// TIA Portal project "Projet_Convoyeurs_S7_1200_Soluce" (V15)
// Vorlageprojekt für das Buch mit Zielsystem S7-1200

(* hardware
DEVICE "S7-1200-Station_1"  S7-1200 Station
   slot 0: "Baugruppenträger_0"  Rack  V1.0
   slot 1: "PLC_1"  CPU 1211C DC/DC/DC  6ES7 211-1AE40-0XB0  V4.1
*)

// ===== PLC "PLC_1"  CPU 1211C DC/DC/DC =====

VAR_GLOBAL   // PLC tag table "Table variables standard"
   "Convoyeur_1_1_Cellule_Debut" AT %I0.0 : Bool;
   "Convoyeur_1_1_Cellule_Fin" AT %I0.1 : Bool;
   "Convoyeur_1_2_Cellule_Debut" AT %I0.2 : Bool;
   "Convoyeur_1_2_Cellule_Fin" AT %I0.3 : Bool;
   "Convoyeur_1_3_Cellule_Debut" AT %I0.4 : Bool;
   "Convoyeur_1_3_Cellule_Fin" AT %I0.5 : Bool;
   "Convoyeur_2_1_Cellule_Debut" AT %I0.6 : Bool;
   "Convoyeur_2_1_Cellule_Fin" AT %I0.7 : Bool;
   "Convoyeur_2_2_Cellule_Debut" AT %I1.0 : Bool;
   "Convoyeur_2_2_Cellule_Fin" AT %I1.1 : Bool;
   "Convoyeur_2_3_Cellule_Debut" AT %I1.2 : Bool;
   "Convoyeur_2_3_Cellule_Fin" AT %I1.3 : Bool;
   "Convoyeur_3_1_Cellule_Debut" AT %I1.4 : Bool;
   "Convoyeur_3_1_Cellule_Fin" AT %I1.5 : Bool;
   "Convoyeur_3_2_Cellule_Debut" AT %I1.6 : Bool;
   "Convoyeur_3_2_Cellule_Fin" AT %I1.7 : Bool;
   "Convoyeur_3_3_Cellule_Debut" AT %I2.0 : Bool;
   "Convoyeur_3_3_Cellule_Fin" AT %I2.1 : Bool;
   "Convoyeur_4_1_Cellule_Debut" AT %I2.2 : Bool;
   "Convoyeur_4_1_Cellule_Fin" AT %I2.3 : Bool;
   "Convoyeur_4_2_Cellule_Debut" AT %I2.4 : Bool;
   "Convoyeur_4_2_Cellule_Fin" AT %I2.5 : Bool;
   "Convoyeur_4_3_Cellule_Debut" AT %I2.6 : Bool;
   "Convoyeur_4_3_Cellule_Fin" AT %I2.7 : Bool;
   "Convoyeur_4_4_Cellule_Debut" AT %I3.0 : Bool;
   "Convoyeur_4_4_Cellule_Fin" AT %I3.1 : Bool;
   "Convoyeur_5_1_Cellule_Debut" AT %I3.2 : Bool;
   "Convoyeur_5_1_Cellule_Fin" AT %I3.3 : Bool;
   "Convoyeur_5_2_Cellule_Debut" AT %I3.4 : Bool;
   "Convoyeur_5_2_Cellule_Fin" AT %I3.5 : Bool;
   "Convoyeur_1_1_AVANCER" AT %Q0.0 : Bool;
   "Convoyeur_1_2_AVANCER" AT %Q0.1 : Bool;
   "Convoyeur_1_3_AVANCER" AT %Q0.2 : Bool;
   "Convoyeur_2_1_AVANCER" AT %Q0.3 : Bool;
   "Convoyeur_2_2_AVANCER" AT %Q0.4 : Bool;
   "Convoyeur_2_3_AVANCER" AT %Q0.5 : Bool;
   "Convoyeur_3_1_AVANCER" AT %Q0.6 : Bool;
   "Convoyeur_3_2_AVANCER" AT %Q0.7 : Bool;
   "Convoyeur_3_3_AVANCER" AT %Q1.0 : Bool;
   "Convoyeur_4_1_AVANCER" AT %Q1.1 : Bool;
   "Convoyeur_4_2_AVANCER" AT %Q1.2 : Bool;
   "Convoyeur_4_3_AVANCER" AT %Q1.3 : Bool;
   "Convoyeur_4_4_AVANCER" AT %Q1.4 : Bool;
   "Convoyeur_5_1_AVANCER" AT %Q1.5 : Bool;
   "Convoyeur_5_2_AVANCER" AT %Q1.6 : Bool;
   "Convoyeur_5_3_AVANCER" AT %Q1.7 : Bool;
   "Convoyeur_5_4_AVANCER" AT %Q2.0 : Bool;
   "Table_1_4_AVANCER" AT %Q2.1 : Bool;
   "Table_1_4_TOURNER_DROITE" AT %Q2.2 : Bool;
   "Table_1_4_TOURNER_GAUCHE" AT %Q2.3 : Bool;
   "Table_1_5_AVANCER" AT %Q2.4 : Bool;
   "Table_1_5_TOURNER_DROITE" AT %Q2.5 : Bool;
   "Table_1_5_TOURNER_GAUCHE" AT %Q2.6 : Bool;
   "Table_2_4_AVANCER" AT %Q2.7 : Bool;
   "Table_2_4_TOURNER_DROITE" AT %Q3.0 : Bool;
   "Table_2_4_TOURNER_GAUCHE" AT %Q3.1 : Bool;
   "Table_2_5_AVANCER" AT %Q3.2 : Bool;
   "Table_2_5_TOURNER_DROITE" AT %Q3.3 : Bool;
   "Table_2_5_TOURNER_GAUCHE" AT %Q3.4 : Bool;
   "Table_3_4_AVANCER" AT %Q3.5 : Bool;
   "Table_3_4_TOURNER_GAUCHE" AT %Q3.7 : Bool;
   "Table_3_4_TOURNER_DROITE" AT %Q3.6 : Bool;
   "Table_3_5_AVANCER" AT %Q4.0 : Bool;
   "Table_3_5_TOURNER_DROITE" AT %Q4.1 : Bool;
   "Table_3_5_TOURNER_GAUCHE" AT %Q4.2 : Bool;
   "Convoyeur_5_3_Cellule_Debut" AT %I3.6 : Bool;
   "Convoyeur_5_3_Cellule_Fin" AT %I3.7 : Bool;
   "Convoyeur_5_4_Cellule_Debut" AT %I4.0 : Bool;
   "Convoyeur_5_4_Cellule_Fin" AT %I4.1 : Bool;
   "Table_1_4_Capteur_Fin" AT %I4.2 : Bool;
   "Table_1_4_Capteur_Droite" AT %I4.3 : Bool;
   "Table_1_4_Capteur_Gauche" AT %I4.4 : Bool;
   "Table_1_5_Capteur_Fin" AT %I4.5 : Bool;
   "Table_1_5_Capteur_Droite" AT %I4.6 : Bool;
   "Table_1_5_Capteur_Gauche" AT %I4.7 : Bool;
   "Table_2_4_Capteur_Fin" AT %I5.0 : Bool;
   "Table_2_4_Capteur_Droite" AT %I5.1 : Bool;
   "Table_2_4_Capteur_Gauche" AT %I5.2 : Bool;
   "Table_2_5_Capteur_Fin" AT %I5.3 : Bool;
   "Table_2_5_Capteur_Droite" AT %I5.4 : Bool;
   "Table_2_5_Capteur_Gauche" AT %I5.5 : Bool;
   "Table_3_4_Capteur_Fin" AT %I5.6 : Bool;
   "Table_3_4_Capteur_Droite" AT %I5.7 : Bool;
   "Table_3_4_Capteur_Gauche" AT %I6.0 : Bool;
   "Table_3_5_Capteur_Fin" AT %I6.1 : Bool;
   "Table_3_5_Capteur_Droite" AT %I6.2 : Bool;
   "Table_3_5_Capteur_Gauche" AT %I6.3 : Bool;
   "Nombre_Total_Ligne_1" AT %QW50 : Int;
   "Nombre_Total_Ligne_2" AT %QW52 : Int;
   "Nombre_Total_Ligne_3" AT %QW54 : Int;
   "Nombre_Total_Ligne_4" AT %QW56 : Int;
   "Nombre_Total_Ligne_5" AT %QW58 : Int;
END_VAR

// folder: DB_Convoyeurs

DATA_BLOCK "Convoyeur_1_1"   // DB3
{ S7_Optimized_Access := 'TRUE' }
VERSION : 0.1
// stored: InstanceOfName Commande_Convoyeur
"Commande_Convoyeur"
BEGIN
END_DATA_BLOCK

DATA_BLOCK "Convoyeur_1_2"   // DB4
{ S7_Optimized_Access := 'TRUE' }
VERSION : 0.1
// stored: InstanceOfName Commande_Convoyeur
"Commande_Convoyeur"
BEGIN
END_DATA_BLOCK

DATA_BLOCK "Convoyeur_4_3"   // DB5
{ S7_Optimized_Access := 'TRUE' }
VERSION : 0.1
// stored: InstanceOfName Commande_Convoyeur
"Commande_Convoyeur"
BEGIN
END_DATA_BLOCK

DATA_BLOCK "Convoyeur_1_3"   // DB6
{ S7_Optimized_Access := 'TRUE' }
VERSION : 0.1
// stored: InstanceOfName Commande_Convoyeur
"Commande_Convoyeur"
BEGIN
END_DATA_BLOCK

DATA_BLOCK "Convoyeur_4_4"   // DB7
{ S7_Optimized_Access := 'TRUE' }
VERSION : 0.1
// stored: InstanceOfName Commande_Convoyeur
"Commande_Convoyeur"
BEGIN
END_DATA_BLOCK

DATA_BLOCK "Convoyeur_5_4"   // DB8
{ S7_Optimized_Access := 'TRUE' }
VERSION : 0.1
// stored: InstanceOfName Commande_Convoyeur
"Commande_Convoyeur"
BEGIN
END_DATA_BLOCK

DATA_BLOCK "Convoyeur_5_3"   // DB9
{ S7_Optimized_Access := 'TRUE' }
VERSION : 0.1
// stored: InstanceOfName Commande_Convoyeur
"Commande_Convoyeur"
BEGIN
END_DATA_BLOCK

DATA_BLOCK "Convoyeur_2_1"   // DB10
{ S7_Optimized_Access := 'TRUE' }
VERSION : 0.1
// stored: InstanceOfName Commande_Convoyeur
"Commande_Convoyeur"
BEGIN
END_DATA_BLOCK

DATA_BLOCK "Convoyeur_2_2"   // DB12
{ S7_Optimized_Access := 'TRUE' }
VERSION : 0.1
// stored: InstanceOfName Commande_Convoyeur
"Commande_Convoyeur"
BEGIN
END_DATA_BLOCK

DATA_BLOCK "Convoyeur_2_3"   // DB14
{ S7_Optimized_Access := 'TRUE' }
VERSION : 0.1
// stored: InstanceOfName Commande_Convoyeur
"Commande_Convoyeur"
BEGIN
END_DATA_BLOCK

DATA_BLOCK "Convoyeur_4_2"   // DB15
{ S7_Optimized_Access := 'TRUE' }
VERSION : 0.1
// stored: InstanceOfName Commande_Convoyeur
"Commande_Convoyeur"
BEGIN
END_DATA_BLOCK

DATA_BLOCK "Convoyeur_5_2"   // DB16
{ S7_Optimized_Access := 'TRUE' }
VERSION : 0.1
// stored: InstanceOfName Commande_Convoyeur
"Commande_Convoyeur"
BEGIN
END_DATA_BLOCK

DATA_BLOCK "Convoyeur_3_1"   // DB19
{ S7_Optimized_Access := 'TRUE' }
VERSION : 0.1
// stored: InstanceOfName Commande_Convoyeur
"Commande_Convoyeur"
BEGIN
END_DATA_BLOCK

DATA_BLOCK "Convoyeur_3_2"   // DB20
{ S7_Optimized_Access := 'TRUE' }
VERSION : 0.1
// stored: InstanceOfName Commande_Convoyeur
"Commande_Convoyeur"
BEGIN
END_DATA_BLOCK

DATA_BLOCK "Convoyeur_3_3"   // DB21
{ S7_Optimized_Access := 'TRUE' }
VERSION : 0.1
// stored: InstanceOfName Commande_Convoyeur
"Commande_Convoyeur"
BEGIN
END_DATA_BLOCK

DATA_BLOCK "Convoyeur_4_1"   // DB22
{ S7_Optimized_Access := 'TRUE' }
VERSION : 0.1
// stored: InstanceOfName Commande_Convoyeur
"Commande_Convoyeur"
BEGIN
END_DATA_BLOCK

DATA_BLOCK "Convoyeur_5_1"   // DB23
{ S7_Optimized_Access := 'TRUE' }
VERSION : 0.1
// stored: InstanceOfName Commande_Convoyeur
"Commande_Convoyeur"
BEGIN
END_DATA_BLOCK

// folder: DB_Tables

DATA_BLOCK "Table_1_4"   // DB1
{ S7_Optimized_Access := 'TRUE' }
VERSION : 0.1
// stored: InstanceOfName Commande_Table
"Commande_Table"
BEGIN
END_DATA_BLOCK

DATA_BLOCK "Table_1_5"   // DB2
{ S7_Optimized_Access := 'TRUE' }
VERSION : 0.1
// stored: InstanceOfName Commande_Table
"Commande_Table"
BEGIN
END_DATA_BLOCK

DATA_BLOCK "Table_2_4"   // DB11
{ S7_Optimized_Access := 'TRUE' }
VERSION : 0.1
// stored: InstanceOfName Commande_Table
"Commande_Table"
BEGIN
END_DATA_BLOCK

DATA_BLOCK "Table_2_5"   // DB13
{ S7_Optimized_Access := 'TRUE' }
VERSION : 0.1
// stored: InstanceOfName Commande_Table
"Commande_Table"
BEGIN
END_DATA_BLOCK

DATA_BLOCK "Table_3_4"   // DB17
{ S7_Optimized_Access := 'TRUE' }
VERSION : 0.1
// stored: InstanceOfName Commande_Table
"Commande_Table"
BEGIN
END_DATA_BLOCK

DATA_BLOCK "Table_3_5"   // DB18
{ S7_Optimized_Access := 'TRUE' }
VERSION : 0.1
// stored: InstanceOfName Commande_Table
"Commande_Table"
BEGIN
END_DATA_BLOCK

// folder: (top level)

FUNCTION_BLOCK "Commande_Table"   // FB1, LAD
{ S7_Optimized_Access := 'TRUE' }
VERSION : 0.1
   VAR_INPUT
      Arrivee_Gauche : Bool;
      Arrivee_Droite : Bool;
      Capteur_Gauche : Bool;
      Capteur_Droite : Bool;
      Capteur_Fin_Table : Bool;
      Evacuation_en_service : Bool;
      Capteur_Debut_Convoyeur_Aval_Gauche : Bool;
      Capteur_Debut_Convoyeur_Aval_Droite : Bool;
   END_VAR
   VAR_OUTPUT
      TOURNER_GAUCHE : Bool;
      TOURNER_DROITE : Bool;
      AVANCER : Bool;
   END_VAR
   VAR
      Etape_GRAFCET : Int;
      Occupee : Bool;
      Priorite_Gauche : Bool;
   END_VAR
BEGIN

REGION Network 1 (SCL): GRAFCET de controle de la table tournante
   CASE #Etape_GRAFCET OF
       0:  // Attente arrivée d'une caisse soit à gauche soit à droite
           IF (#Arrivee_Gauche AND ((NOT #Arrivee_Droite) OR (#Arrivee_Droite AND #Priorite_Gauche))) THEN
               #Etape_GRAFCET := 1;
           END_IF;
           IF (#Arrivee_Droite AND ((NOT #Arrivee_Gauche) OR (#Arrivee_Gauche AND (NOT #Priorite_Gauche)))) THEN
               #Etape_GRAFCET := 2;
           END_IF;
       1:  // Tourner vers la gauche
           IF #Capteur_Gauche THEN
               #Etape_GRAFCET := 3;
           END_IF;
       2:  // Tourner vers la droite
           IF #Capteur_Droite THEN
               #Etape_GRAFCET := 3;
           END_IF;
       3:  // Avance de la caisse jusqu'à la fin de la table
           IF (#Capteur_Fin_Table AND (NOT #Evacuation_en_service)) THEN
               #Etape_GRAFCET := 4;
           END_IF;
           IF (#Capteur_Fin_Table AND #Evacuation_en_service) THEN
               #Etape_GRAFCET := 5;
           END_IF;
       4:  // Arrêt et Attente évacuation en service
           IF #Evacuation_en_service THEN
               #Etape_GRAFCET := 5;
           END_IF;
       5:  // Evacuation de la caisse
           IF (NOT #Capteur_Fin_Table) THEN
               #Etape_GRAFCET := 6;
           END_IF;
       6:  // Fin Evacuation de la caisse
           IF ((#Capteur_Gauche AND (NOT #Capteur_Debut_Convoyeur_Aval_Gauche)) OR (#Capteur_Droite AND (NOT #Capteur_Debut_Convoyeur_Aval_Droite))) THEN
               #Etape_GRAFCET := 0;
           END_IF;
       ELSE
           #Etape_GRAFCET := 0;
   END_CASE;
END_REGION

REGION Network 2: Commande des sorties
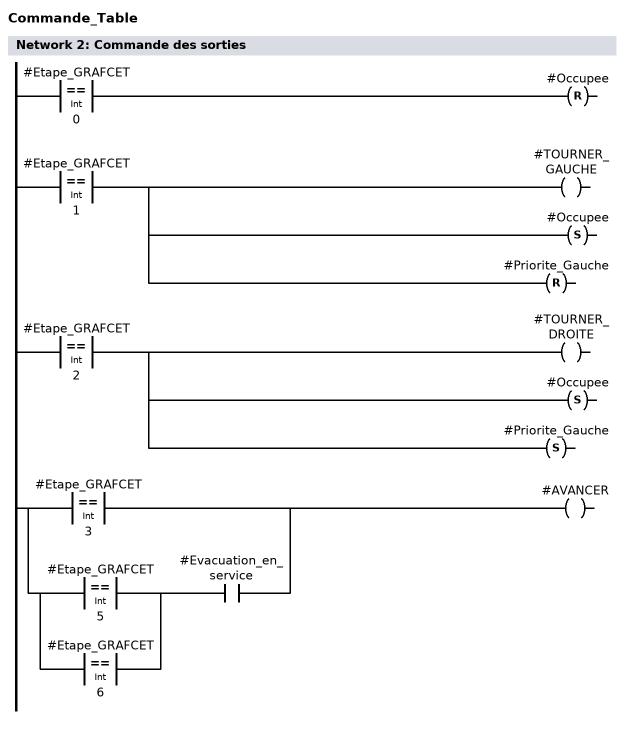
   RUNG wire#powerrail
      { S7_Templates := "SrcType := Int" } EQ_Contact(in1 := #Etape_GRAFCET, in2 := 0)
      R_Coil( #Occupee )
   END_RUNG
   RUNG wire#powerrail
      { S7_Templates := "SrcType := Int" } EQ_Contact(in1 := #Etape_GRAFCET, in2 := 1)
      wire#w1
      Coil( #TOURNER_GAUCHE )
   END_RUNG
   RUNG wire#w1
      S_Coil( #Occupee )
   END_RUNG
   RUNG wire#w1
      R_Coil( #Priorite_Gauche )
   END_RUNG
   RUNG wire#powerrail
      { S7_Templates := "SrcType := Int" } EQ_Contact(in1 := #Etape_GRAFCET, in2 := 2)
      wire#w2
      Coil( #TOURNER_DROITE )
   END_RUNG
   RUNG wire#w2
      S_Coil( #Occupee )
   END_RUNG
   RUNG wire#w2
      S_Coil( #Priorite_Gauche )
   END_RUNG
   RUNG wire#powerrail
      { S7_Templates := "SrcType := Int" } EQ_Contact(in1 := #Etape_GRAFCET, in2 := 3)
      wire#w3
      Coil( #AVANCER )
   END_RUNG
   RUNG wire#powerrail
      { S7_Templates := "SrcType := Int" } EQ_Contact(in1 := #Etape_GRAFCET, in2 := 5)
      wire#w4
      Contact( #Evacuation_en_service )
   END_RUNG wire#w3
   RUNG wire#powerrail
      { S7_Templates := "SrcType := Int" } EQ_Contact(in1 := #Etape_GRAFCET, in2 := 6)
   END_RUNG wire#w4
   // the same network as SCL:
   IF #Etape_GRAFCET = 0 THEN #Occupee := FALSE; END_IF;
   #TOURNER_GAUCHE := #Etape_GRAFCET = 1;
   IF #TOURNER_GAUCHE THEN
       #Occupee := TRUE;
       #Priorite_Gauche := FALSE;
   END_IF;
   #TOURNER_DROITE := #Etape_GRAFCET = 2;
   IF #TOURNER_DROITE THEN
       #Occupee := TRUE;
       #Priorite_Gauche := TRUE;
   END_IF;
   #AVANCER := (#Etape_GRAFCET = 3) OR (((#Etape_GRAFCET = 5) OR (#Etape_GRAFCET = 6)) AND #Evacuation_en_service);
END_REGION
END_FUNCTION_BLOCK

FUNCTION_BLOCK "Commande_Convoyeur"   // FB2, LAD
{ S7_Optimized_Access := 'TRUE' }
VERSION : 0.1
   VAR_INPUT
      Capteur_Debut_Convoyeur : Bool;
      Capteur_Fin_Convoyeur : Bool;
      Etape_Grafcet_Table : Int;
      Table_Bonne_Direction : Bool;
      Fin_Table_Amont : Bool;
      Terminaison : Bool;
   END_VAR
   VAR_OUTPUT
      AVANCER : Bool;
   END_VAR
   VAR
      Etape_GRAFCET : Int;
      Nombre_Caisses : Int;
      Nombre_Caisses_Total : Int;
      Front_Capteur_Debut : Bool;
      Front_Capteur_Fin : Bool;
   END_VAR
   VAR_TEMP   // added for the SCL form of the ladder/FBD networks
      _w1 : Bool;
      _w2 : Bool;
   END_VAR
BEGIN

REGION Network 1: Comptage Caisses
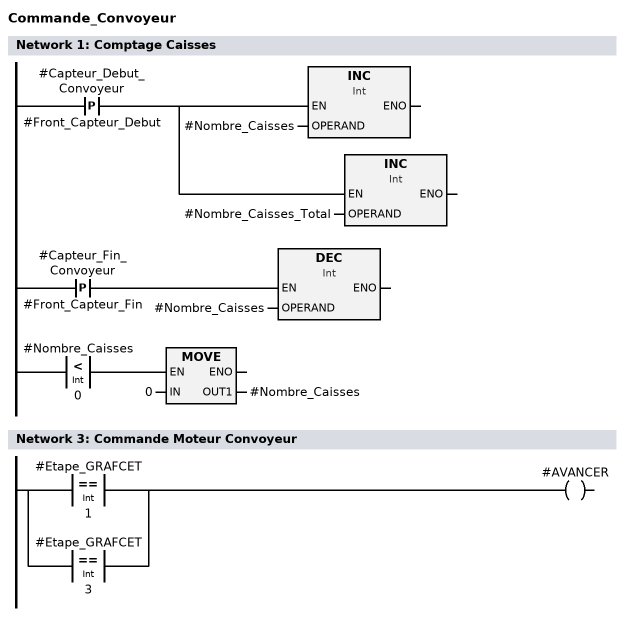
   RUNG wire#powerrail
      P_Contact(operand := #Capteur_Debut_Convoyeur, bit := #Front_Capteur_Debut)
      wire#w1
      { S7_Templates := "DestType := Int" } Inc( #Nombre_Caisses )
   END_RUNG
   RUNG wire#w1
      { S7_Templates := "DestType := Int" } Inc( #Nombre_Caisses_Total )
   END_RUNG
   RUNG wire#powerrail
      P_Contact(operand := #Capteur_Fin_Convoyeur, bit := #Front_Capteur_Fin)
      { S7_Templates := "DestType := Int" } Dec( #Nombre_Caisses )
   END_RUNG
   RUNG wire#powerrail
      { S7_Templates := "SrcType := Int" } LT_Contact(in1 := #Nombre_Caisses, in2 := 0)
      Move(in := 0, out1 => #Nombre_Caisses)
   END_RUNG
   // the same network as SCL:
   #_w1 := #Capteur_Debut_Convoyeur AND NOT #Front_Capteur_Debut;   // rising edge of #Capteur_Debut_Convoyeur
   #Front_Capteur_Debut := #Capteur_Debut_Convoyeur;
   IF #_w1 THEN
       #Nombre_Caisses := #Nombre_Caisses + 1;
       #Nombre_Caisses_Total := #Nombre_Caisses_Total + 1;
   END_IF;
   #_w2 := #Capteur_Fin_Convoyeur AND NOT #Front_Capteur_Fin;   // rising edge of #Capteur_Fin_Convoyeur
   #Front_Capteur_Fin := #Capteur_Fin_Convoyeur;
   IF #_w2 THEN #Nombre_Caisses := #Nombre_Caisses - 1; END_IF;
   IF #Nombre_Caisses < 0 THEN #Nombre_Caisses := 0; END_IF;
END_REGION

REGION Network 2 (SCL): GRAFCET de controle d'un convoyeur
   CASE #Etape_GRAFCET OF
       0:  // Attente ordre départ
           IF ((#Nombre_Caisses>0) OR ((#Nombre_Caisses=0)AND #Fin_Table_Amont))  THEN
               #Etape_GRAFCET := 1;
           END_IF;
       1:  // Avance jusqu'au capteur de fin
           IF #Capteur_Fin_Convoyeur THEN
               #Etape_GRAFCET := 2;
           END_IF;
       2:  // Arret - Attente table bonne direction et Debut chargement table
           IF (#Table_Bonne_Direction AND (#Etape_Grafcet_Table = 3)) THEN
               #Etape_GRAFCET := 3;
           END_IF;
       3:  // Avance jusqu'à chargement table terminé
           IF (NOT #Capteur_Fin_Convoyeur) THEN
               #Etape_GRAFCET := 4;
           END_IF;
       4:  // Arret - Attente fin évacuation table
           IF ((#Table_Bonne_Direction AND (#Etape_Grafcet_Table = 6))OR #Terminaison) THEN
               #Etape_GRAFCET := 0;
           END_IF;
       ELSE  
           #Etape_GRAFCET := 0;
   END_CASE;
END_REGION

REGION Network 3: Commande Moteur Convoyeur
   RUNG wire#powerrail
      { S7_Templates := "SrcType := Int" } EQ_Contact(in1 := #Etape_GRAFCET, in2 := 1)
      wire#w1
      Coil( #AVANCER )
   END_RUNG
   RUNG wire#powerrail
      { S7_Templates := "SrcType := Int" } EQ_Contact(in1 := #Etape_GRAFCET, in2 := 3)
   END_RUNG wire#w1
   // the same network as SCL:
   #AVANCER := (#Etape_GRAFCET = 1) OR (#Etape_GRAFCET = 3);
END_REGION
END_FUNCTION_BLOCK

FUNCTION "MHJ-PLC-Lab-Function-S71200" : Void   // FC9000, SCL
{ S7_Optimized_Access := 'TRUE' }
VERSION : 0.1
   VAR_TEMP
      rdTimeReturn : Int;
      outputTime : DTL;
      SyncVal : Byte;
      forVal : Int;
      forVal_2 : Int;
      Value : Byte;
   END_VAR
   VAR CONSTANT
      CompVal : Byte := 16#34;
      Value_01 : Byte := 16#11;
      Value_01_DW : DWord := 16#A165_D992;
      Value_02_DW : DWord := 16#58BE_4401;
   END_VAR
BEGIN

   #Value:=PEEK(area := 16#82,
        dbNumber := 0,
        byteOffset := 511);
   #Value := #Value + 1;

   POKE(area := 16#82,
        dbNumber := 0,
        byteOffset := 511,
        value := #Value);

   POKE(area:=16#81,
        dbNumber:=0,
        byteOffset:=1016,
        value:=#Value_01_DW);
   POKE(area := 16#81,
        dbNumber := 0,
        byteOffset := 1020,
        value := #Value_02_DW);

   POKE(area := 16#81,
        dbNumber := 0,
        byteOffset := 511,
        value := B#16#00);

   FOR #forVal := 0 TO 120 DO
       FOR #forVal_2:=0 TO 10 DO
           #rdTimeReturn:=RD_SYS_T(#outputTime);
           #rdTimeReturn := WR_SYS_T(#outputTime);
           #rdTimeReturn := RD_SYS_T(#outputTime);
           #rdTimeReturn := WR_SYS_T(#outputTime);
       END_FOR;
       #SyncVal:= PEEK(area := 16#81,
                      dbNumber := 0,
                      byteOffset := 511);
       IF #SyncVal = #CompVal THEN
          GOTO M_1;
       END_IF;
   END_FOR;
   RETURN;

   M_1:
   POKE(area := 16#81,
        dbNumber := 0,
        byteOffset := 511,
        value := B#16#0);
END_FUNCTION

ORGANIZATION_BLOCK "Main"   // OB1, LAD, ProgramCycle
TITLE = "Main Program Sweep (Cycle)"
{ S7_Optimized_Access := 'TRUE' }
VERSION : 0.1
   VAR_INPUT
      Initial_Call : Bool;   // Initial call of this OB
      Remanence : Bool;   // =True, if remanent data are available
   END_VAR
BEGIN

REGION Network 1: Konnektierungsbaustein für PLC-Lab / Appel Fonction MHJ pour Factory-IO
   // Im Netzwerk 1 wird der Konnektierungsbaustein für PLC-Lab aufgerufen.
   // Dieser Aufruf darf nicht entfernt werden!
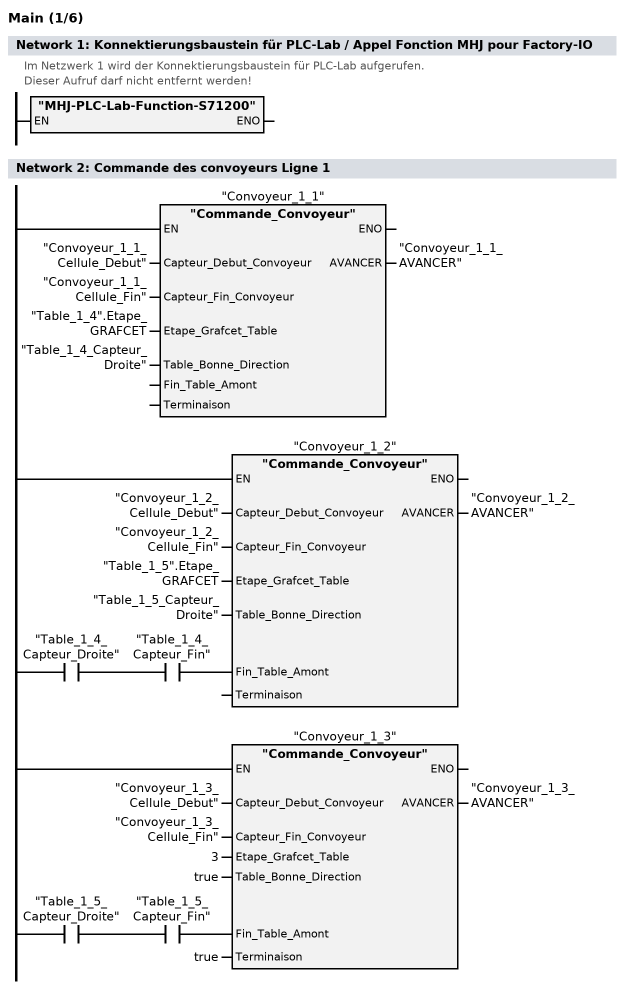
   RUNG wire#powerrail
      "MHJ-PLC-Lab-Function-S71200"()
   END_RUNG
   // the same network as SCL:
   "MHJ-PLC-Lab-Function-S71200"();
END_REGION

REGION Network 2: Commande des convoyeurs Ligne 1
   RUNG wire#powerrail
      "Convoyeur_1_1"(Capteur_Debut_Convoyeur := "Convoyeur_1_1_Cellule_Debut", Capteur_Fin_Convoyeur := "Convoyeur_1_1_Cellule_Fin", Etape_Grafcet_Table := "Table_1_4".Etape_GRAFCET, Table_Bonne_Direction := "Table_1_4_Capteur_Droite", Fin_Table_Amont :=, Terminaison :=, AVANCER => "Convoyeur_1_1_AVANCER")
   END_RUNG
   RUNG wire#powerrail
      "Convoyeur_1_2"(Fin_Table_Amont := wire#w1, Capteur_Debut_Convoyeur := "Convoyeur_1_2_Cellule_Debut", Capteur_Fin_Convoyeur := "Convoyeur_1_2_Cellule_Fin", Etape_Grafcet_Table := "Table_1_5".Etape_GRAFCET, Table_Bonne_Direction := "Table_1_5_Capteur_Droite", Terminaison :=, AVANCER => "Convoyeur_1_2_AVANCER")
   END_RUNG
   RUNG wire#powerrail
      Contact( "Table_1_4_Capteur_Droite" )
      Contact( "Table_1_4_Capteur_Fin" )
   END_RUNG wire#w1
   RUNG wire#powerrail
      "Convoyeur_1_3"(Fin_Table_Amont := wire#w2, Capteur_Debut_Convoyeur := "Convoyeur_1_3_Cellule_Debut", Capteur_Fin_Convoyeur := "Convoyeur_1_3_Cellule_Fin", Etape_Grafcet_Table := 3, Table_Bonne_Direction := true, Terminaison := true, AVANCER => "Convoyeur_1_3_AVANCER")
   END_RUNG
   RUNG wire#powerrail
      Contact( "Table_1_5_Capteur_Droite" )
      Contact( "Table_1_5_Capteur_Fin" )
   END_RUNG wire#w2
   // the same network as SCL:
   "Convoyeur_1_1"(Capteur_Debut_Convoyeur := "Convoyeur_1_1_Cellule_Debut",   // "Commande_Convoyeur"
                   Capteur_Fin_Convoyeur := "Convoyeur_1_1_Cellule_Fin",
                   Etape_Grafcet_Table := "Table_1_4".Etape_GRAFCET,
                   Table_Bonne_Direction := "Table_1_4_Capteur_Droite",
                   AVANCER => "Convoyeur_1_1_AVANCER");
   "Convoyeur_1_2"(Capteur_Debut_Convoyeur := "Convoyeur_1_2_Cellule_Debut",   // "Commande_Convoyeur"
                   Capteur_Fin_Convoyeur := "Convoyeur_1_2_Cellule_Fin",
                   Etape_Grafcet_Table := "Table_1_5".Etape_GRAFCET,
                   Table_Bonne_Direction := "Table_1_5_Capteur_Droite",
                   Fin_Table_Amont := "Table_1_4_Capteur_Droite" AND "Table_1_4_Capteur_Fin",
                   AVANCER => "Convoyeur_1_2_AVANCER");
   "Convoyeur_1_3"(Capteur_Debut_Convoyeur := "Convoyeur_1_3_Cellule_Debut",   // "Commande_Convoyeur"
                   Capteur_Fin_Convoyeur := "Convoyeur_1_3_Cellule_Fin",
                   Etape_Grafcet_Table := 3,
                   Table_Bonne_Direction := true,
                   Fin_Table_Amont := "Table_1_5_Capteur_Droite" AND "Table_1_5_Capteur_Fin",
                   Terminaison := true,
                   AVANCER => "Convoyeur_1_3_AVANCER");
END_REGION

REGION Network 3: Commande des convoyeurs Ligne 2
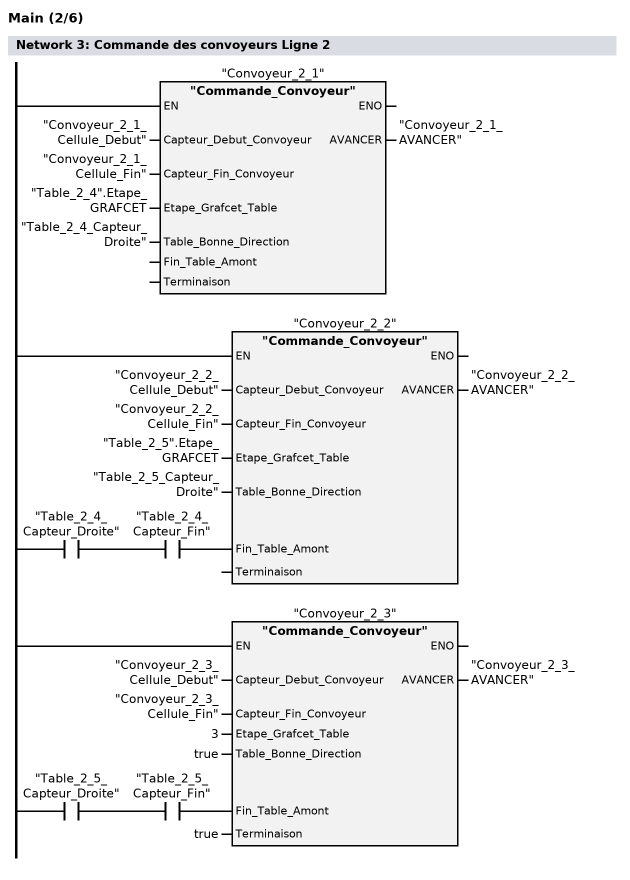
   RUNG wire#powerrail
      "Convoyeur_2_1"(Capteur_Debut_Convoyeur := "Convoyeur_2_1_Cellule_Debut", Capteur_Fin_Convoyeur := "Convoyeur_2_1_Cellule_Fin", Etape_Grafcet_Table := "Table_2_4".Etape_GRAFCET, Table_Bonne_Direction := "Table_2_4_Capteur_Droite", Fin_Table_Amont :=, Terminaison :=, AVANCER => "Convoyeur_2_1_AVANCER")
   END_RUNG
   RUNG wire#powerrail
      "Convoyeur_2_2"(Fin_Table_Amont := wire#w1, Capteur_Debut_Convoyeur := "Convoyeur_2_2_Cellule_Debut", Capteur_Fin_Convoyeur := "Convoyeur_2_2_Cellule_Fin", Etape_Grafcet_Table := "Table_2_5".Etape_GRAFCET, Table_Bonne_Direction := "Table_2_5_Capteur_Droite", Terminaison :=, AVANCER => "Convoyeur_2_2_AVANCER")
   END_RUNG
   RUNG wire#powerrail
      Contact( "Table_2_4_Capteur_Droite" )
      Contact( "Table_2_4_Capteur_Fin" )
   END_RUNG wire#w1
   RUNG wire#powerrail
      "Convoyeur_2_3"(Fin_Table_Amont := wire#w2, Capteur_Debut_Convoyeur := "Convoyeur_2_3_Cellule_Debut", Capteur_Fin_Convoyeur := "Convoyeur_2_3_Cellule_Fin", Etape_Grafcet_Table := 3, Table_Bonne_Direction := true, Terminaison := true, AVANCER => "Convoyeur_2_3_AVANCER")
   END_RUNG
   RUNG wire#powerrail
      Contact( "Table_2_5_Capteur_Droite" )
      Contact( "Table_2_5_Capteur_Fin" )
   END_RUNG wire#w2
   // the same network as SCL:
   "Convoyeur_2_1"(Capteur_Debut_Convoyeur := "Convoyeur_2_1_Cellule_Debut",   // "Commande_Convoyeur"
                   Capteur_Fin_Convoyeur := "Convoyeur_2_1_Cellule_Fin",
                   Etape_Grafcet_Table := "Table_2_4".Etape_GRAFCET,
                   Table_Bonne_Direction := "Table_2_4_Capteur_Droite",
                   AVANCER => "Convoyeur_2_1_AVANCER");
   "Convoyeur_2_2"(Capteur_Debut_Convoyeur := "Convoyeur_2_2_Cellule_Debut",   // "Commande_Convoyeur"
                   Capteur_Fin_Convoyeur := "Convoyeur_2_2_Cellule_Fin",
                   Etape_Grafcet_Table := "Table_2_5".Etape_GRAFCET,
                   Table_Bonne_Direction := "Table_2_5_Capteur_Droite",
                   Fin_Table_Amont := "Table_2_4_Capteur_Droite" AND "Table_2_4_Capteur_Fin",
                   AVANCER => "Convoyeur_2_2_AVANCER");
   "Convoyeur_2_3"(Capteur_Debut_Convoyeur := "Convoyeur_2_3_Cellule_Debut",   // "Commande_Convoyeur"
                   Capteur_Fin_Convoyeur := "Convoyeur_2_3_Cellule_Fin",
                   Etape_Grafcet_Table := 3,
                   Table_Bonne_Direction := true,
                   Fin_Table_Amont := "Table_2_5_Capteur_Droite" AND "Table_2_5_Capteur_Fin",
                   Terminaison := true,
                   AVANCER => "Convoyeur_2_3_AVANCER");
END_REGION

REGION Network 4: Commande des convoyeurs Ligne 3
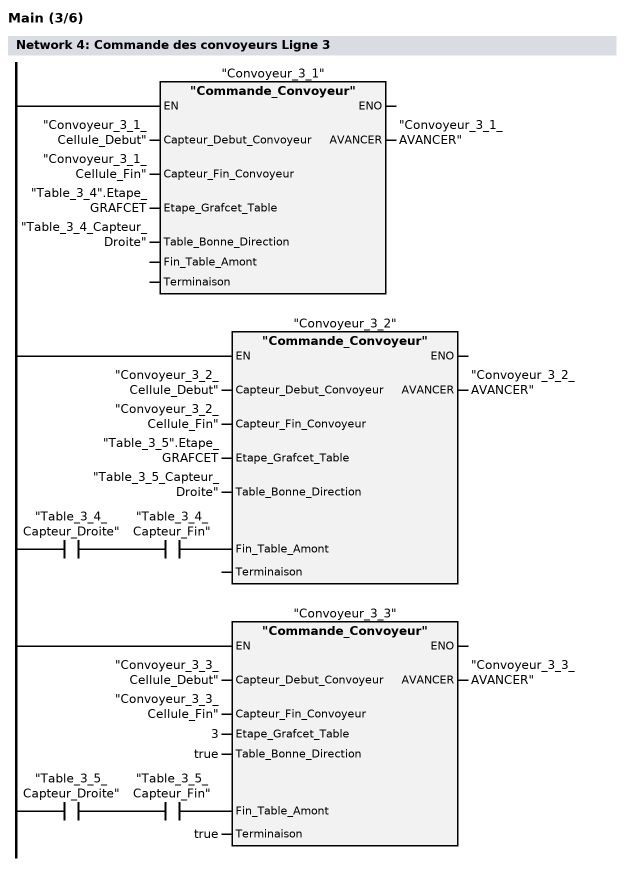
   RUNG wire#powerrail
      "Convoyeur_3_1"(Capteur_Debut_Convoyeur := "Convoyeur_3_1_Cellule_Debut", Capteur_Fin_Convoyeur := "Convoyeur_3_1_Cellule_Fin", Etape_Grafcet_Table := "Table_3_4".Etape_GRAFCET, Table_Bonne_Direction := "Table_3_4_Capteur_Droite", Fin_Table_Amont :=, Terminaison :=, AVANCER => "Convoyeur_3_1_AVANCER")
   END_RUNG
   RUNG wire#powerrail
      "Convoyeur_3_2"(Fin_Table_Amont := wire#w1, Capteur_Debut_Convoyeur := "Convoyeur_3_2_Cellule_Debut", Capteur_Fin_Convoyeur := "Convoyeur_3_2_Cellule_Fin", Etape_Grafcet_Table := "Table_3_5".Etape_GRAFCET, Table_Bonne_Direction := "Table_3_5_Capteur_Droite", Terminaison :=, AVANCER => "Convoyeur_3_2_AVANCER")
   END_RUNG
   RUNG wire#powerrail
      Contact( "Table_3_4_Capteur_Droite" )
      Contact( "Table_3_4_Capteur_Fin" )
   END_RUNG wire#w1
   RUNG wire#powerrail
      "Convoyeur_3_3"(Fin_Table_Amont := wire#w2, Capteur_Debut_Convoyeur := "Convoyeur_3_3_Cellule_Debut", Capteur_Fin_Convoyeur := "Convoyeur_3_3_Cellule_Fin", Etape_Grafcet_Table := 3, Table_Bonne_Direction := true, Terminaison := true, AVANCER => "Convoyeur_3_3_AVANCER")
   END_RUNG
   RUNG wire#powerrail
      Contact( "Table_3_5_Capteur_Droite" )
      Contact( "Table_3_5_Capteur_Fin" )
   END_RUNG wire#w2
   // the same network as SCL:
   "Convoyeur_3_1"(Capteur_Debut_Convoyeur := "Convoyeur_3_1_Cellule_Debut",   // "Commande_Convoyeur"
                   Capteur_Fin_Convoyeur := "Convoyeur_3_1_Cellule_Fin",
                   Etape_Grafcet_Table := "Table_3_4".Etape_GRAFCET,
                   Table_Bonne_Direction := "Table_3_4_Capteur_Droite",
                   AVANCER => "Convoyeur_3_1_AVANCER");
   "Convoyeur_3_2"(Capteur_Debut_Convoyeur := "Convoyeur_3_2_Cellule_Debut",   // "Commande_Convoyeur"
                   Capteur_Fin_Convoyeur := "Convoyeur_3_2_Cellule_Fin",
                   Etape_Grafcet_Table := "Table_3_5".Etape_GRAFCET,
                   Table_Bonne_Direction := "Table_3_5_Capteur_Droite",
                   Fin_Table_Amont := "Table_3_4_Capteur_Droite" AND "Table_3_4_Capteur_Fin",
                   AVANCER => "Convoyeur_3_2_AVANCER");
   "Convoyeur_3_3"(Capteur_Debut_Convoyeur := "Convoyeur_3_3_Cellule_Debut",   // "Commande_Convoyeur"
                   Capteur_Fin_Convoyeur := "Convoyeur_3_3_Cellule_Fin",
                   Etape_Grafcet_Table := 3,
                   Table_Bonne_Direction := true,
                   Fin_Table_Amont := "Table_3_5_Capteur_Droite" AND "Table_3_5_Capteur_Fin",
                   Terminaison := true,
                   AVANCER => "Convoyeur_3_3_AVANCER");
END_REGION

REGION Network 5: Commande des convoyeurs Ligne 4
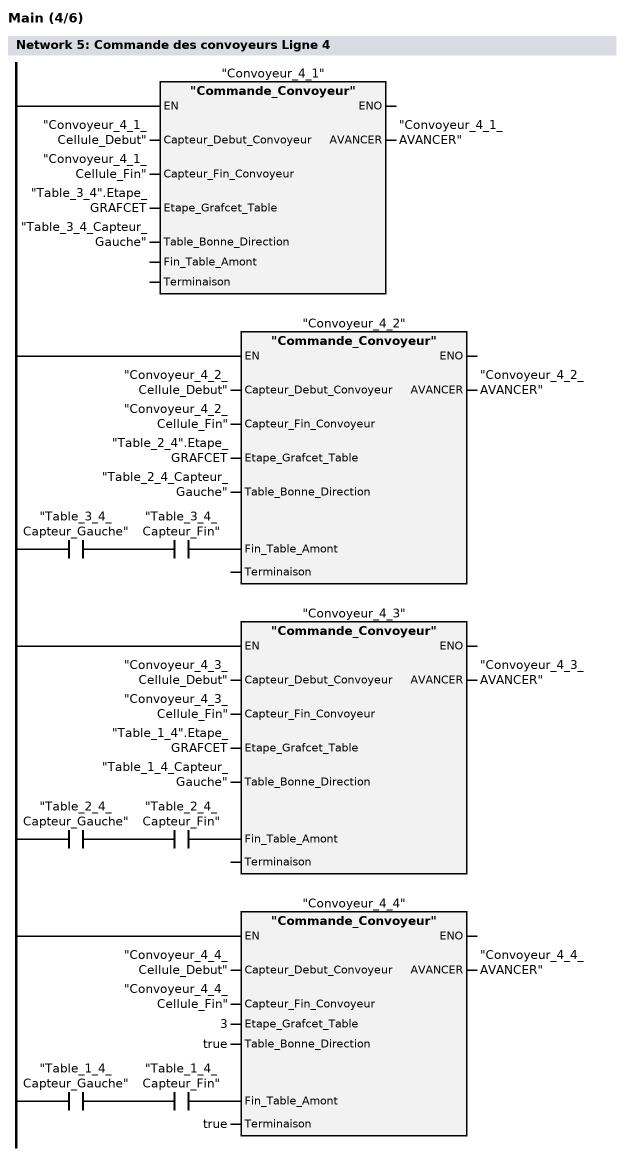
   RUNG wire#powerrail
      "Convoyeur_4_1"(Capteur_Debut_Convoyeur := "Convoyeur_4_1_Cellule_Debut", Capteur_Fin_Convoyeur := "Convoyeur_4_1_Cellule_Fin", Etape_Grafcet_Table := "Table_3_4".Etape_GRAFCET, Table_Bonne_Direction := "Table_3_4_Capteur_Gauche", Fin_Table_Amont :=, Terminaison :=, AVANCER => "Convoyeur_4_1_AVANCER")
   END_RUNG
   RUNG wire#powerrail
      "Convoyeur_4_2"(Fin_Table_Amont := wire#w1, Capteur_Debut_Convoyeur := "Convoyeur_4_2_Cellule_Debut", Capteur_Fin_Convoyeur := "Convoyeur_4_2_Cellule_Fin", Etape_Grafcet_Table := "Table_2_4".Etape_GRAFCET, Table_Bonne_Direction := "Table_2_4_Capteur_Gauche", Terminaison :=, AVANCER => "Convoyeur_4_2_AVANCER")
   END_RUNG
   RUNG wire#powerrail
      Contact( "Table_3_4_Capteur_Gauche" )
      Contact( "Table_3_4_Capteur_Fin" )
   END_RUNG wire#w1
   RUNG wire#powerrail
      "Convoyeur_4_3"(Fin_Table_Amont := wire#w2, Capteur_Debut_Convoyeur := "Convoyeur_4_3_Cellule_Debut", Capteur_Fin_Convoyeur := "Convoyeur_4_3_Cellule_Fin", Etape_Grafcet_Table := "Table_1_4".Etape_GRAFCET, Table_Bonne_Direction := "Table_1_4_Capteur_Gauche", Terminaison :=, AVANCER => "Convoyeur_4_3_AVANCER")
   END_RUNG
   RUNG wire#powerrail
      Contact( "Table_2_4_Capteur_Gauche" )
      Contact( "Table_2_4_Capteur_Fin" )
   END_RUNG wire#w2
   RUNG wire#powerrail
      "Convoyeur_4_4"(Fin_Table_Amont := wire#w3, Capteur_Debut_Convoyeur := "Convoyeur_4_4_Cellule_Debut", Capteur_Fin_Convoyeur := "Convoyeur_4_4_Cellule_Fin", Etape_Grafcet_Table := 3, Table_Bonne_Direction := true, Terminaison := true, AVANCER => "Convoyeur_4_4_AVANCER")
   END_RUNG
   RUNG wire#powerrail
      Contact( "Table_1_4_Capteur_Gauche" )
      Contact( "Table_1_4_Capteur_Fin" )
   END_RUNG wire#w3
   // the same network as SCL:
   "Convoyeur_4_1"(Capteur_Debut_Convoyeur := "Convoyeur_4_1_Cellule_Debut",   // "Commande_Convoyeur"
                   Capteur_Fin_Convoyeur := "Convoyeur_4_1_Cellule_Fin",
                   Etape_Grafcet_Table := "Table_3_4".Etape_GRAFCET,
                   Table_Bonne_Direction := "Table_3_4_Capteur_Gauche",
                   AVANCER => "Convoyeur_4_1_AVANCER");
   "Convoyeur_4_2"(Capteur_Debut_Convoyeur := "Convoyeur_4_2_Cellule_Debut",   // "Commande_Convoyeur"
                   Capteur_Fin_Convoyeur := "Convoyeur_4_2_Cellule_Fin",
                   Etape_Grafcet_Table := "Table_2_4".Etape_GRAFCET,
                   Table_Bonne_Direction := "Table_2_4_Capteur_Gauche",
                   Fin_Table_Amont := "Table_3_4_Capteur_Gauche" AND "Table_3_4_Capteur_Fin",
                   AVANCER => "Convoyeur_4_2_AVANCER");
   "Convoyeur_4_3"(Capteur_Debut_Convoyeur := "Convoyeur_4_3_Cellule_Debut",   // "Commande_Convoyeur"
                   Capteur_Fin_Convoyeur := "Convoyeur_4_3_Cellule_Fin",
                   Etape_Grafcet_Table := "Table_1_4".Etape_GRAFCET,
                   Table_Bonne_Direction := "Table_1_4_Capteur_Gauche",
                   Fin_Table_Amont := "Table_2_4_Capteur_Gauche" AND "Table_2_4_Capteur_Fin",
                   AVANCER => "Convoyeur_4_3_AVANCER");
   "Convoyeur_4_4"(Capteur_Debut_Convoyeur := "Convoyeur_4_4_Cellule_Debut",   // "Commande_Convoyeur"
                   Capteur_Fin_Convoyeur := "Convoyeur_4_4_Cellule_Fin",
                   Etape_Grafcet_Table := 3,
                   Table_Bonne_Direction := true,
                   Fin_Table_Amont := "Table_1_4_Capteur_Gauche" AND "Table_1_4_Capteur_Fin",
                   Terminaison := true,
                   AVANCER => "Convoyeur_4_4_AVANCER");
END_REGION

REGION Network 6: Commande des convoyeurs Ligne 5
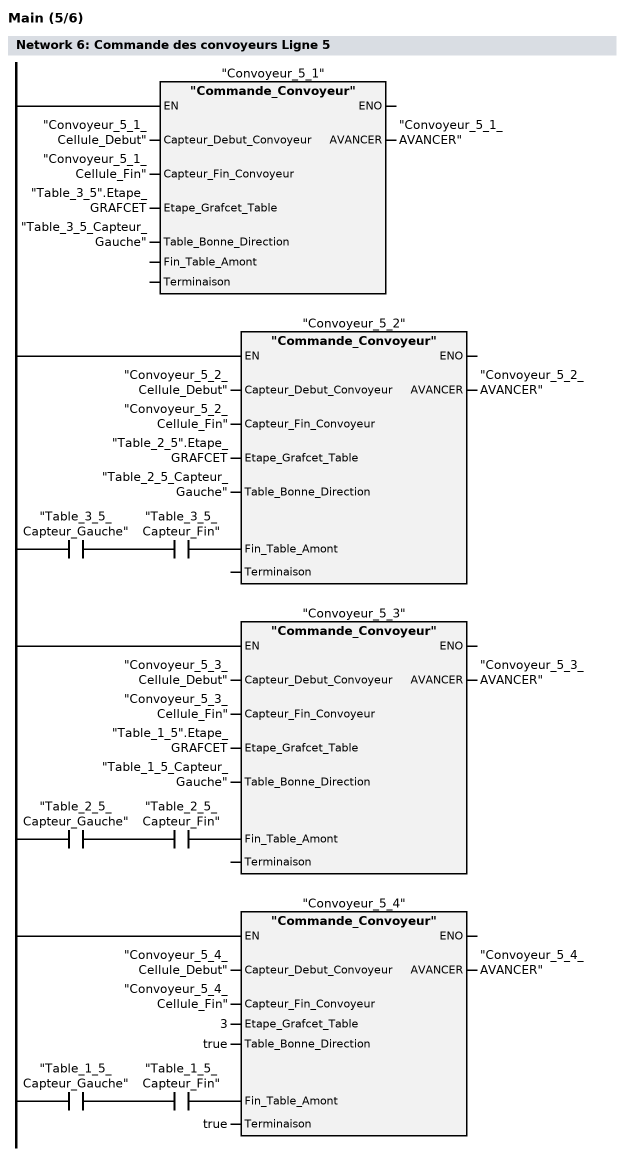
   RUNG wire#powerrail
      "Convoyeur_5_1"(Capteur_Debut_Convoyeur := "Convoyeur_5_1_Cellule_Debut", Capteur_Fin_Convoyeur := "Convoyeur_5_1_Cellule_Fin", Etape_Grafcet_Table := "Table_3_5".Etape_GRAFCET, Table_Bonne_Direction := "Table_3_5_Capteur_Gauche", Fin_Table_Amont :=, Terminaison :=, AVANCER => "Convoyeur_5_1_AVANCER")
   END_RUNG
   RUNG wire#powerrail
      "Convoyeur_5_2"(Fin_Table_Amont := wire#w1, Capteur_Debut_Convoyeur := "Convoyeur_5_2_Cellule_Debut", Capteur_Fin_Convoyeur := "Convoyeur_5_2_Cellule_Fin", Etape_Grafcet_Table := "Table_2_5".Etape_GRAFCET, Table_Bonne_Direction := "Table_2_5_Capteur_Gauche", Terminaison :=, AVANCER => "Convoyeur_5_2_AVANCER")
   END_RUNG
   RUNG wire#powerrail
      Contact( "Table_3_5_Capteur_Gauche" )
      Contact( "Table_3_5_Capteur_Fin" )
   END_RUNG wire#w1
   RUNG wire#powerrail
      "Convoyeur_5_3"(Fin_Table_Amont := wire#w2, Capteur_Debut_Convoyeur := "Convoyeur_5_3_Cellule_Debut", Capteur_Fin_Convoyeur := "Convoyeur_5_3_Cellule_Fin", Etape_Grafcet_Table := "Table_1_5".Etape_GRAFCET, Table_Bonne_Direction := "Table_1_5_Capteur_Gauche", Terminaison :=, AVANCER => "Convoyeur_5_3_AVANCER")
   END_RUNG
   RUNG wire#powerrail
      Contact( "Table_2_5_Capteur_Gauche" )
      Contact( "Table_2_5_Capteur_Fin" )
   END_RUNG wire#w2
   RUNG wire#powerrail
      "Convoyeur_5_4"(Fin_Table_Amont := wire#w3, Capteur_Debut_Convoyeur := "Convoyeur_5_4_Cellule_Debut", Capteur_Fin_Convoyeur := "Convoyeur_5_4_Cellule_Fin", Etape_Grafcet_Table := 3, Table_Bonne_Direction := true, Terminaison := true, AVANCER => "Convoyeur_5_4_AVANCER")
   END_RUNG
   RUNG wire#powerrail
      Contact( "Table_1_5_Capteur_Gauche" )
      Contact( "Table_1_5_Capteur_Fin" )
   END_RUNG wire#w3
   // the same network as SCL:
   "Convoyeur_5_1"(Capteur_Debut_Convoyeur := "Convoyeur_5_1_Cellule_Debut",   // "Commande_Convoyeur"
                   Capteur_Fin_Convoyeur := "Convoyeur_5_1_Cellule_Fin",
                   Etape_Grafcet_Table := "Table_3_5".Etape_GRAFCET,
                   Table_Bonne_Direction := "Table_3_5_Capteur_Gauche",
                   AVANCER => "Convoyeur_5_1_AVANCER");
   "Convoyeur_5_2"(Capteur_Debut_Convoyeur := "Convoyeur_5_2_Cellule_Debut",   // "Commande_Convoyeur"
                   Capteur_Fin_Convoyeur := "Convoyeur_5_2_Cellule_Fin",
                   Etape_Grafcet_Table := "Table_2_5".Etape_GRAFCET,
                   Table_Bonne_Direction := "Table_2_5_Capteur_Gauche",
                   Fin_Table_Amont := "Table_3_5_Capteur_Gauche" AND "Table_3_5_Capteur_Fin",
                   AVANCER => "Convoyeur_5_2_AVANCER");
   "Convoyeur_5_3"(Capteur_Debut_Convoyeur := "Convoyeur_5_3_Cellule_Debut",   // "Commande_Convoyeur"
                   Capteur_Fin_Convoyeur := "Convoyeur_5_3_Cellule_Fin",
                   Etape_Grafcet_Table := "Table_1_5".Etape_GRAFCET,
                   Table_Bonne_Direction := "Table_1_5_Capteur_Gauche",
                   Fin_Table_Amont := "Table_2_5_Capteur_Gauche" AND "Table_2_5_Capteur_Fin",
                   AVANCER => "Convoyeur_5_3_AVANCER");
   "Convoyeur_5_4"(Capteur_Debut_Convoyeur := "Convoyeur_5_4_Cellule_Debut",   // "Commande_Convoyeur"
                   Capteur_Fin_Convoyeur := "Convoyeur_5_4_Cellule_Fin",
                   Etape_Grafcet_Table := 3,
                   Table_Bonne_Direction := true,
                   Fin_Table_Amont := "Table_1_5_Capteur_Gauche" AND "Table_1_5_Capteur_Fin",
                   Terminaison := true,
                   AVANCER => "Convoyeur_5_4_AVANCER");
END_REGION

REGION Network 7: Commande des tables tournantes
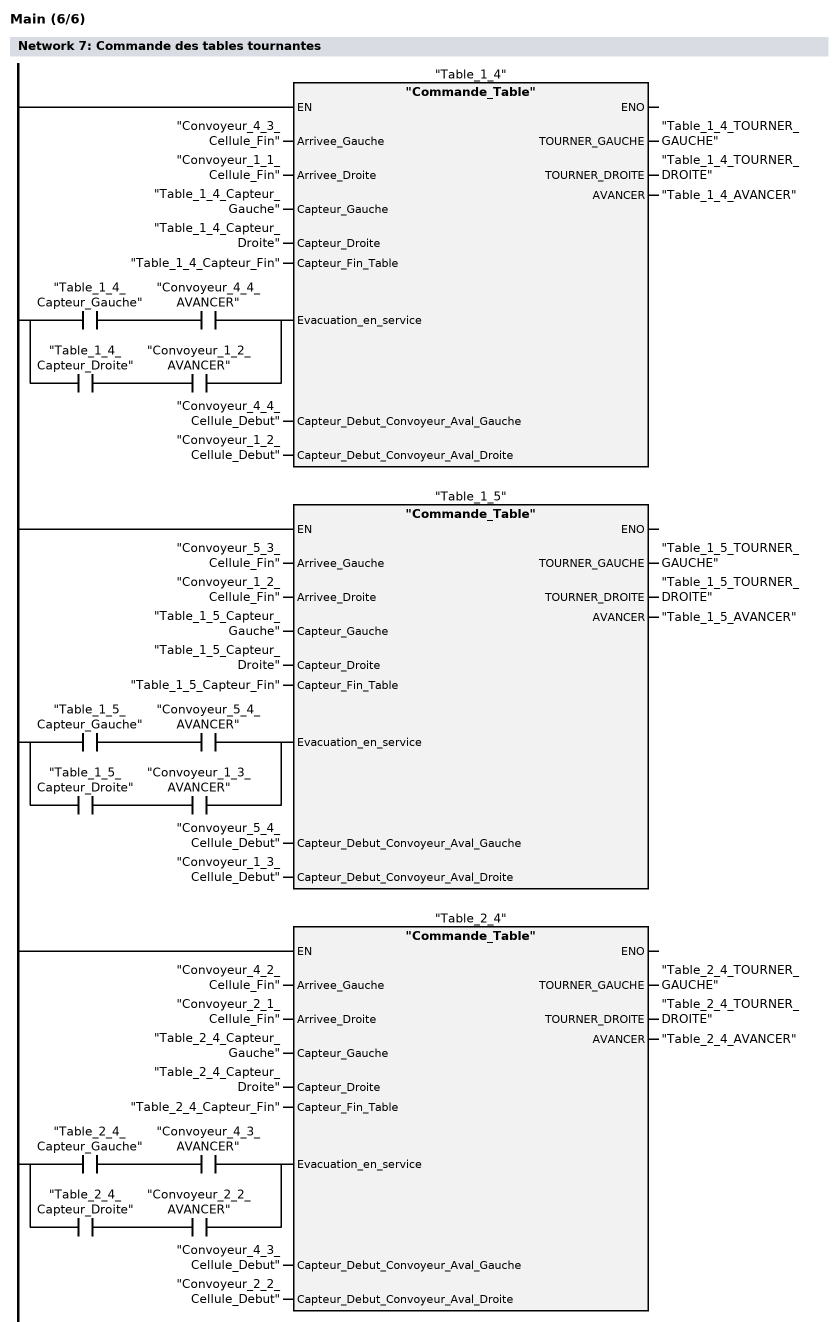
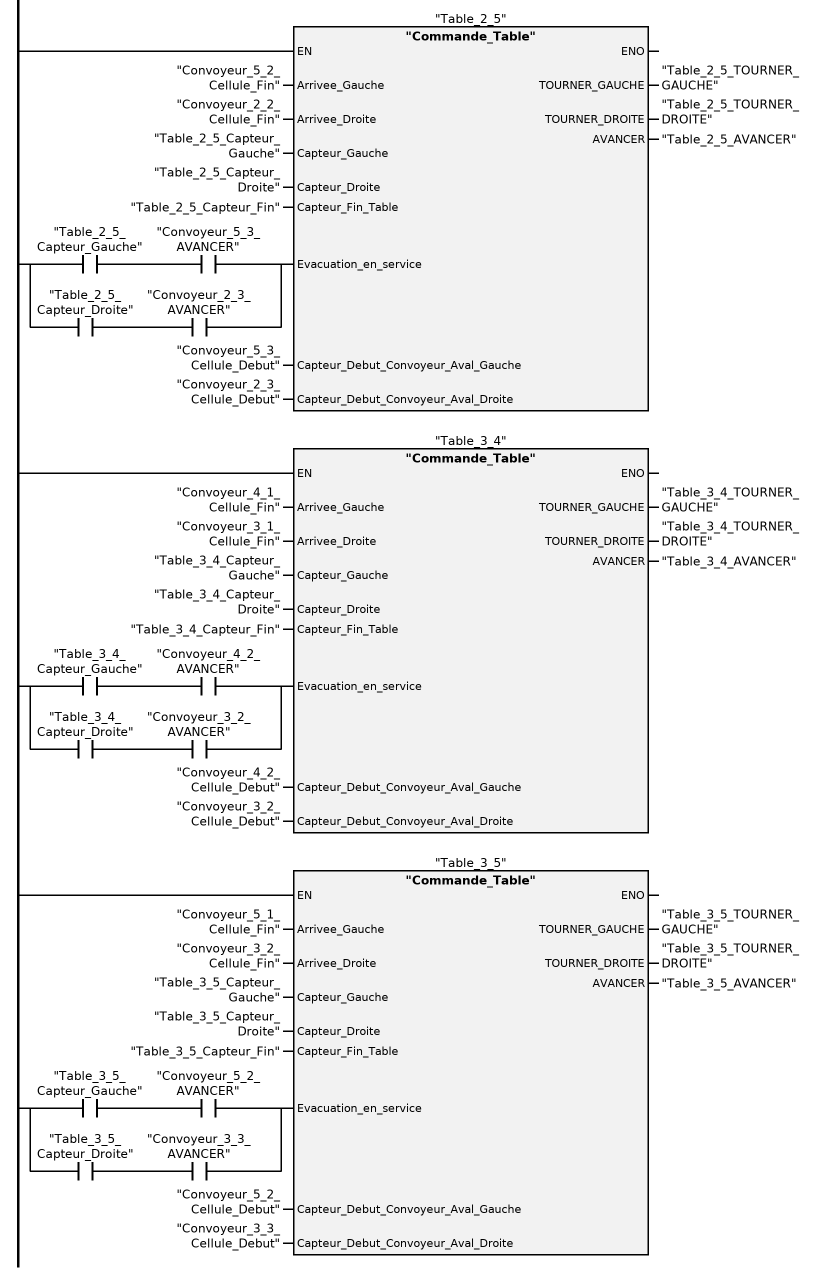
   RUNG wire#powerrail
      "Table_1_4"(Evacuation_en_service := wire#w1, Arrivee_Gauche := "Convoyeur_4_3_Cellule_Fin", Arrivee_Droite := "Convoyeur_1_1_Cellule_Fin", Capteur_Gauche := "Table_1_4_Capteur_Gauche", Capteur_Droite := "Table_1_4_Capteur_Droite", Capteur_Fin_Table := "Table_1_4_Capteur_Fin", Capteur_Debut_Convoyeur_Aval_Gauche := "Convoyeur_4_4_Cellule_Debut", Capteur_Debut_Convoyeur_Aval_Droite := "Convoyeur_1_2_Cellule_Debut", TOURNER_GAUCHE => "Table_1_4_TOURNER_GAUCHE", TOURNER_DROITE => "Table_1_4_TOURNER_DROITE", AVANCER => "Table_1_4_AVANCER")
   END_RUNG
   RUNG wire#powerrail
      Contact( "Table_1_4_Capteur_Gauche" )
      Contact( "Convoyeur_4_4_AVANCER" )
   END_RUNG wire#w1
   RUNG wire#powerrail
      Contact( "Table_1_4_Capteur_Droite" )
      Contact( "Convoyeur_1_2_AVANCER" )
   END_RUNG wire#w1
   RUNG wire#powerrail
      "Table_1_5"(Evacuation_en_service := wire#w2, Arrivee_Gauche := "Convoyeur_5_3_Cellule_Fin", Arrivee_Droite := "Convoyeur_1_2_Cellule_Fin", Capteur_Gauche := "Table_1_5_Capteur_Gauche", Capteur_Droite := "Table_1_5_Capteur_Droite", Capteur_Fin_Table := "Table_1_5_Capteur_Fin", Capteur_Debut_Convoyeur_Aval_Gauche := "Convoyeur_5_4_Cellule_Debut", Capteur_Debut_Convoyeur_Aval_Droite := "Convoyeur_1_3_Cellule_Debut", TOURNER_GAUCHE => "Table_1_5_TOURNER_GAUCHE", TOURNER_DROITE => "Table_1_5_TOURNER_DROITE", AVANCER => "Table_1_5_AVANCER")
   END_RUNG
   RUNG wire#powerrail
      Contact( "Table_1_5_Capteur_Gauche" )
      Contact( "Convoyeur_5_4_AVANCER" )
   END_RUNG wire#w2
   RUNG wire#powerrail
      Contact( "Table_1_5_Capteur_Droite" )
      Contact( "Convoyeur_1_3_AVANCER" )
   END_RUNG wire#w2
   RUNG wire#powerrail
      "Table_2_4"(Evacuation_en_service := wire#w3, Arrivee_Gauche := "Convoyeur_4_2_Cellule_Fin", Arrivee_Droite := "Convoyeur_2_1_Cellule_Fin", Capteur_Gauche := "Table_2_4_Capteur_Gauche", Capteur_Droite := "Table_2_4_Capteur_Droite", Capteur_Fin_Table := "Table_2_4_Capteur_Fin", Capteur_Debut_Convoyeur_Aval_Gauche := "Convoyeur_4_3_Cellule_Debut", Capteur_Debut_Convoyeur_Aval_Droite := "Convoyeur_2_2_Cellule_Debut", TOURNER_GAUCHE => "Table_2_4_TOURNER_GAUCHE", TOURNER_DROITE => "Table_2_4_TOURNER_DROITE", AVANCER => "Table_2_4_AVANCER")
   END_RUNG
   RUNG wire#powerrail
      Contact( "Table_2_4_Capteur_Gauche" )
      Contact( "Convoyeur_4_3_AVANCER" )
   END_RUNG wire#w3
   RUNG wire#powerrail
      Contact( "Table_2_4_Capteur_Droite" )
      Contact( "Convoyeur_2_2_AVANCER" )
   END_RUNG wire#w3
   RUNG wire#powerrail
      "Table_2_5"(Evacuation_en_service := wire#w4, Arrivee_Gauche := "Convoyeur_5_2_Cellule_Fin", Arrivee_Droite := "Convoyeur_2_2_Cellule_Fin", Capteur_Gauche := "Table_2_5_Capteur_Gauche", Capteur_Droite := "Table_2_5_Capteur_Droite", Capteur_Fin_Table := "Table_2_5_Capteur_Fin", Capteur_Debut_Convoyeur_Aval_Gauche := "Convoyeur_5_3_Cellule_Debut", Capteur_Debut_Convoyeur_Aval_Droite := "Convoyeur_2_3_Cellule_Debut", TOURNER_GAUCHE => "Table_2_5_TOURNER_GAUCHE", TOURNER_DROITE => "Table_2_5_TOURNER_DROITE", AVANCER => "Table_2_5_AVANCER")
   END_RUNG
   RUNG wire#powerrail
      Contact( "Table_2_5_Capteur_Gauche" )
      Contact( "Convoyeur_5_3_AVANCER" )
   END_RUNG wire#w4
   RUNG wire#powerrail
      Contact( "Table_2_5_Capteur_Droite" )
      Contact( "Convoyeur_2_3_AVANCER" )
   END_RUNG wire#w4
   RUNG wire#powerrail
      "Table_3_4"(Evacuation_en_service := wire#w5, Arrivee_Gauche := "Convoyeur_4_1_Cellule_Fin", Arrivee_Droite := "Convoyeur_3_1_Cellule_Fin", Capteur_Gauche := "Table_3_4_Capteur_Gauche", Capteur_Droite := "Table_3_4_Capteur_Droite", Capteur_Fin_Table := "Table_3_4_Capteur_Fin", Capteur_Debut_Convoyeur_Aval_Gauche := "Convoyeur_4_2_Cellule_Debut", Capteur_Debut_Convoyeur_Aval_Droite := "Convoyeur_3_2_Cellule_Debut", TOURNER_GAUCHE => "Table_3_4_TOURNER_GAUCHE", TOURNER_DROITE => "Table_3_4_TOURNER_DROITE", AVANCER => "Table_3_4_AVANCER")
   END_RUNG
   RUNG wire#powerrail
      Contact( "Table_3_4_Capteur_Gauche" )
      Contact( "Convoyeur_4_2_AVANCER" )
   END_RUNG wire#w5
   RUNG wire#powerrail
      Contact( "Table_3_4_Capteur_Droite" )
      Contact( "Convoyeur_3_2_AVANCER" )
   END_RUNG wire#w5
   RUNG wire#powerrail
      "Table_3_5"(Evacuation_en_service := wire#w6, Arrivee_Gauche := "Convoyeur_5_1_Cellule_Fin", Arrivee_Droite := "Convoyeur_3_2_Cellule_Fin", Capteur_Gauche := "Table_3_5_Capteur_Gauche", Capteur_Droite := "Table_3_5_Capteur_Droite", Capteur_Fin_Table := "Table_3_5_Capteur_Fin", Capteur_Debut_Convoyeur_Aval_Gauche := "Convoyeur_5_2_Cellule_Debut", Capteur_Debut_Convoyeur_Aval_Droite := "Convoyeur_3_3_Cellule_Debut", TOURNER_GAUCHE => "Table_3_5_TOURNER_GAUCHE", TOURNER_DROITE => "Table_3_5_TOURNER_DROITE", AVANCER => "Table_3_5_AVANCER")
   END_RUNG
   RUNG wire#powerrail
      Contact( "Table_3_5_Capteur_Gauche" )
      Contact( "Convoyeur_5_2_AVANCER" )
   END_RUNG wire#w6
   RUNG wire#powerrail
      Contact( "Table_3_5_Capteur_Droite" )
      Contact( "Convoyeur_3_3_AVANCER" )
   END_RUNG wire#w6
   // the same network as SCL:
   "Table_1_4"(Arrivee_Gauche := "Convoyeur_4_3_Cellule_Fin",   // "Commande_Table"
               Arrivee_Droite := "Convoyeur_1_1_Cellule_Fin",
               Capteur_Gauche := "Table_1_4_Capteur_Gauche",
               Capteur_Droite := "Table_1_4_Capteur_Droite",
               Capteur_Fin_Table := "Table_1_4_Capteur_Fin",
               Evacuation_en_service := ("Table_1_4_Capteur_Gauche" AND "Convoyeur_4_4_AVANCER") OR ("Table_1_4_Capteur_Droite" AND "Convoyeur_1_2_AVANCER"),
               Capteur_Debut_Convoyeur_Aval_Gauche := "Convoyeur_4_4_Cellule_Debut",
               Capteur_Debut_Convoyeur_Aval_Droite := "Convoyeur_1_2_Cellule_Debut",
               TOURNER_GAUCHE => "Table_1_4_TOURNER_GAUCHE",
               TOURNER_DROITE => "Table_1_4_TOURNER_DROITE",
               AVANCER => "Table_1_4_AVANCER");
   "Table_1_5"(Arrivee_Gauche := "Convoyeur_5_3_Cellule_Fin",   // "Commande_Table"
               Arrivee_Droite := "Convoyeur_1_2_Cellule_Fin",
               Capteur_Gauche := "Table_1_5_Capteur_Gauche",
               Capteur_Droite := "Table_1_5_Capteur_Droite",
               Capteur_Fin_Table := "Table_1_5_Capteur_Fin",
               Evacuation_en_service := ("Table_1_5_Capteur_Gauche" AND "Convoyeur_5_4_AVANCER") OR ("Table_1_5_Capteur_Droite" AND "Convoyeur_1_3_AVANCER"),
               Capteur_Debut_Convoyeur_Aval_Gauche := "Convoyeur_5_4_Cellule_Debut",
               Capteur_Debut_Convoyeur_Aval_Droite := "Convoyeur_1_3_Cellule_Debut",
               TOURNER_GAUCHE => "Table_1_5_TOURNER_GAUCHE",
               TOURNER_DROITE => "Table_1_5_TOURNER_DROITE",
               AVANCER => "Table_1_5_AVANCER");
   "Table_2_4"(Arrivee_Gauche := "Convoyeur_4_2_Cellule_Fin",   // "Commande_Table"
               Arrivee_Droite := "Convoyeur_2_1_Cellule_Fin",
               Capteur_Gauche := "Table_2_4_Capteur_Gauche",
               Capteur_Droite := "Table_2_4_Capteur_Droite",
               Capteur_Fin_Table := "Table_2_4_Capteur_Fin",
               Evacuation_en_service := ("Table_2_4_Capteur_Gauche" AND "Convoyeur_4_3_AVANCER") OR ("Table_2_4_Capteur_Droite" AND "Convoyeur_2_2_AVANCER"),
               Capteur_Debut_Convoyeur_Aval_Gauche := "Convoyeur_4_3_Cellule_Debut",
               Capteur_Debut_Convoyeur_Aval_Droite := "Convoyeur_2_2_Cellule_Debut",
               TOURNER_GAUCHE => "Table_2_4_TOURNER_GAUCHE",
               TOURNER_DROITE => "Table_2_4_TOURNER_DROITE",
               AVANCER => "Table_2_4_AVANCER");
   "Table_2_5"(Arrivee_Gauche := "Convoyeur_5_2_Cellule_Fin",   // "Commande_Table"
               Arrivee_Droite := "Convoyeur_2_2_Cellule_Fin",
               Capteur_Gauche := "Table_2_5_Capteur_Gauche",
               Capteur_Droite := "Table_2_5_Capteur_Droite",
               Capteur_Fin_Table := "Table_2_5_Capteur_Fin",
               Evacuation_en_service := ("Table_2_5_Capteur_Gauche" AND "Convoyeur_5_3_AVANCER") OR ("Table_2_5_Capteur_Droite" AND "Convoyeur_2_3_AVANCER"),
               Capteur_Debut_Convoyeur_Aval_Gauche := "Convoyeur_5_3_Cellule_Debut",
               Capteur_Debut_Convoyeur_Aval_Droite := "Convoyeur_2_3_Cellule_Debut",
               TOURNER_GAUCHE => "Table_2_5_TOURNER_GAUCHE",
               TOURNER_DROITE => "Table_2_5_TOURNER_DROITE",
               AVANCER => "Table_2_5_AVANCER");
   "Table_3_4"(Arrivee_Gauche := "Convoyeur_4_1_Cellule_Fin",   // "Commande_Table"
               Arrivee_Droite := "Convoyeur_3_1_Cellule_Fin",
               Capteur_Gauche := "Table_3_4_Capteur_Gauche",
               Capteur_Droite := "Table_3_4_Capteur_Droite",
               Capteur_Fin_Table := "Table_3_4_Capteur_Fin",
               Evacuation_en_service := ("Table_3_4_Capteur_Gauche" AND "Convoyeur_4_2_AVANCER") OR ("Table_3_4_Capteur_Droite" AND "Convoyeur_3_2_AVANCER"),
               Capteur_Debut_Convoyeur_Aval_Gauche := "Convoyeur_4_2_Cellule_Debut",
               Capteur_Debut_Convoyeur_Aval_Droite := "Convoyeur_3_2_Cellule_Debut",
               TOURNER_GAUCHE => "Table_3_4_TOURNER_GAUCHE",
               TOURNER_DROITE => "Table_3_4_TOURNER_DROITE",
               AVANCER => "Table_3_4_AVANCER");
   "Table_3_5"(Arrivee_Gauche := "Convoyeur_5_1_Cellule_Fin",   // "Commande_Table"
               Arrivee_Droite := "Convoyeur_3_2_Cellule_Fin",
               Capteur_Gauche := "Table_3_5_Capteur_Gauche",
               Capteur_Droite := "Table_3_5_Capteur_Droite",
               Capteur_Fin_Table := "Table_3_5_Capteur_Fin",
               Evacuation_en_service := ("Table_3_5_Capteur_Gauche" AND "Convoyeur_5_2_AVANCER") OR ("Table_3_5_Capteur_Droite" AND "Convoyeur_3_3_AVANCER"),
               Capteur_Debut_Convoyeur_Aval_Gauche := "Convoyeur_5_2_Cellule_Debut",
               Capteur_Debut_Convoyeur_Aval_Droite := "Convoyeur_3_3_Cellule_Debut",
               TOURNER_GAUCHE => "Table_3_5_TOURNER_GAUCHE",
               TOURNER_DROITE => "Table_3_5_TOURNER_DROITE",
               AVANCER => "Table_3_5_AVANCER");
END_REGION

REGION Network 8 (SCL): Affichage des nombres de caisses sur PO - Totaux fin de ligne
   "Nombre_Total_Ligne_1" := "Convoyeur_1_3".Nombre_Caisses_Total;
   "Nombre_Total_Ligne_2" := "Convoyeur_2_3".Nombre_Caisses_Total;
   "Nombre_Total_Ligne_3" := "Convoyeur_3_3".Nombre_Caisses_Total;
   "Nombre_Total_Ligne_4" := "Convoyeur_4_4".Nombre_Caisses_Total;
   "Nombre_Total_Ligne_5" := "Convoyeur_5_4".Nombre_Caisses_Total;
END_REGION
END_ORGANIZATION_BLOCK